PROGRAM PRG_LI2K2_K2A
VAR
    {attribute 'pytmc' := '
        pv: LI2K2:K2A
        io: io
    '}
    fbLI2K2: FB_LIC;

    //stSiBP: ST_BeamParams := PMPS_GVL.cstFullBeam;
    //stFoilBP: ST_BeamParams := PMPS_GVL.cstFullBeam;
END_VAR

(*
   Avoid damage peak between 3.2 keV and 1.6 keV
*)
//stSiBp.neVRange := F_eVExcludeRange(1600, 3200);
// Drop transmission to 20%
//stSiBP.nTran := 0.2;

// Drop transmission to 10%
////stFoilBP.nTran := 0.1;

fbLI2K2.stOut.fPosition := 1.2;
fbLI2K2.stOut.bUseRawCounts := FALSE;
fbLI2K2.stOut.bValid := TRUE;
fbLI2K2.stOut.stPMPS.sPmpsState := 'LI2K2:K2A-OUT';

fbLI2K2.stMirror1.fPosition := -35.3;
fbLI2K2.stMirror1.bUseRawCounts := FALSE;
fbLI2K2.stMirror1.bValid := TRUE;
fbLI2K2.stMirror1.stPMPS.sPmpsState := 'LI2K2:K2A-MIRROR1';

fbLI2K2.stMirror2.fPosition := -69.3;
fbLI2K2.stMirror2.bUseRawCounts := FALSE;
fbLI2K2.stMirror2.bValid := TRUE;
fbLI2K2.stMirror2.stPMPS.sPmpsState := 'LI2K2:K2A-MIRROR2';

fbLI2K2.stTarget1.fPosition := -101.3;
fbLI2K2.stTarget1.bUseRawCounts := FALSE;
fbLI2K2.stTarget1.bValid := TRUE;
fbLI2K2.stTarget1.stPMPS.sPmpsState := 'LI2K2:K2A-TARGET1';

fbLI2K2(
    fbArbiter := GVL.fbArbiter2,
    fbFFHWO := GVL.fbFastFaultOutput2,
    stYStage := Main.M11,
    sDeviceName := 'LI2K2:K2A',
    sTransitionKey := 'LI2K2:K2A-TRANSITION',
    bEnableMotion := TRUE,
    bEnableBeamParams := TRUE,
    bEnablePositionLimits := TRUE,
);

END_PROGRAM

(* stored: Version 1.1.0.1, ProductVersion 3.1.4022.18
   POU PRG_LI2K2_K2A: Id {9ffb2115-7d48-4e03-8278-7e55d55de1e7}, SpecialFunc None *)
